// TIA Portal project "1200S7PLC_RS485ModBus_OPCUA" (V19)

(* hardware
DEVICE "S7-1200 station_1"  S7-1200 Station
   slot 0: "Rack_0"  S7-1200 Rack  Rack  V1.0
   slot 1: "PLC_1"  CPU 1212C DC/DC/Rly  6ES7 212-1HE40-0XB0  V4.6
   slot 3: "CB 1241 (RS485)"  CB 1241 (RS485)  6ES7 241-1CH30-1XB0  V1.0
*)

// ===== PLC "PLC_1"  CPU 1212C DC/DC/Rly =====

VAR_GLOBAL   // PLC tag table "Default tag table"
   "System_Byte" AT %MB500 : Byte;
   "FirstScan" AT %M500.0 : Bool;
   "DiagStatusUpdate" AT %M500.1 : Bool;
   "AlwaysTRUE" AT %M500.2 : Bool;
   "AlwaysFALSE" AT %M500.3 : Bool;
   "Clock_Byte" AT %MB501 : Byte;
   "Clock_10Hz" AT %M501.0 : Bool;
   "Clock_5Hz" AT %M501.1 : Bool;
   "Clock_2.5Hz" AT %M501.2 : Bool;
   "Clock_2Hz" AT %M501.3 : Bool;
   "Clock_1.25Hz" AT %M501.4 : Bool;
   "Clock_1Hz" AT %M501.5 : Bool;
   "Clock_0.625Hz" AT %M501.6 : Bool;
   "Clock_0.5Hz" AT %M501.7 : Bool;
   "COMM_LOAD_DONE" AT %M2.0 : Bool;
   "COMM_LOAD_ERROR" AT %M2.1 : Bool;
   "COMM_LOAD_STATUS" AT %MW4 : Word;
   "MASTER_DONE" AT %M2.2 : Bool;
   "MASTER_BUSY" AT %M2.3 : Bool;
   "MASTER_ERROR" AT %M2.4 : Bool;
   "MASTER_STATUS" AT %MW6 : Word;
   "HumidityRaw" AT %MD8 : Real;
   "HumidityReal" AT %MD12 : Real;
   "TemperatureRaw" AT %MD16 : Real;
   "TemperatureReal" AT %MD20 : Real;
END_VAR

DATA_BLOCK "ModbusReadData"   // DB3
{ S7_Optimized_Access := 'FALSE' }
VERSION : 0.1
   VAR
      ModbusSensorData : Array[0..1] of Int;
   END_VAR
BEGIN
END_DATA_BLOCK

FUNCTION "Conversion" : Void   // FC1, LAD
{ S7_Optimized_Access := 'TRUE' }
VERSION : 0.1
BEGIN

REGION Network 1
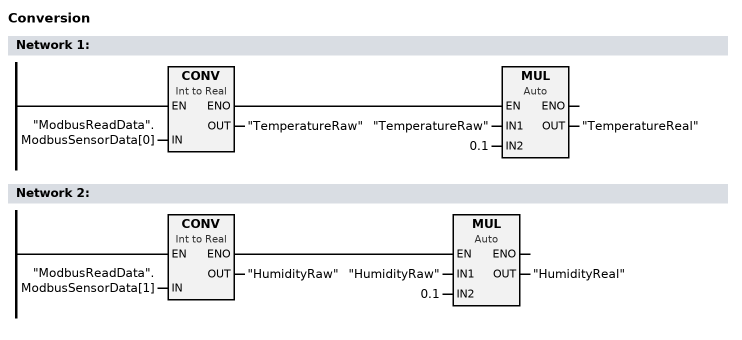
   RUNG wire#powerrail
      { S7_Templates := "[SrcType := Int, DestType := Real]" } Convert(in := "ModbusReadData".ModbusSensorData[0], out => "TemperatureRaw")
      Mul(in1 := "TemperatureRaw", in2 := 0.1, out => "TemperatureReal")
   END_RUNG
   // the same network as SCL:
   "TemperatureRaw" := INT_TO_REAL("ModbusReadData".ModbusSensorData[0]);
   "TemperatureReal" := "TemperatureRaw" * 0.1;
END_REGION

REGION Network 2
   RUNG wire#powerrail
      { S7_Templates := "[SrcType := Int, DestType := Real]" } Convert(in := "ModbusReadData".ModbusSensorData[1], out => "HumidityRaw")
      Mul(in1 := "HumidityRaw", in2 := 0.1, out => "HumidityReal")
   END_RUNG
   // the same network as SCL:
   "HumidityRaw" := INT_TO_REAL("ModbusReadData".ModbusSensorData[1]);
   "HumidityReal" := "HumidityRaw" * 0.1;
END_REGION
END_FUNCTION

ORGANIZATION_BLOCK "Main"   // OB1, LAD, ProgramCycle
TITLE = "Main Program Sweep (Cycle)"
{ S7_Optimized_Access := 'TRUE' }
VERSION : 0.1
   VAR_INPUT
      Initial_Call : Bool;   // Initial call of this OB
      Remanence : Bool;   // =True, if remanent data are available
   END_VAR
BEGIN

REGION Network 1
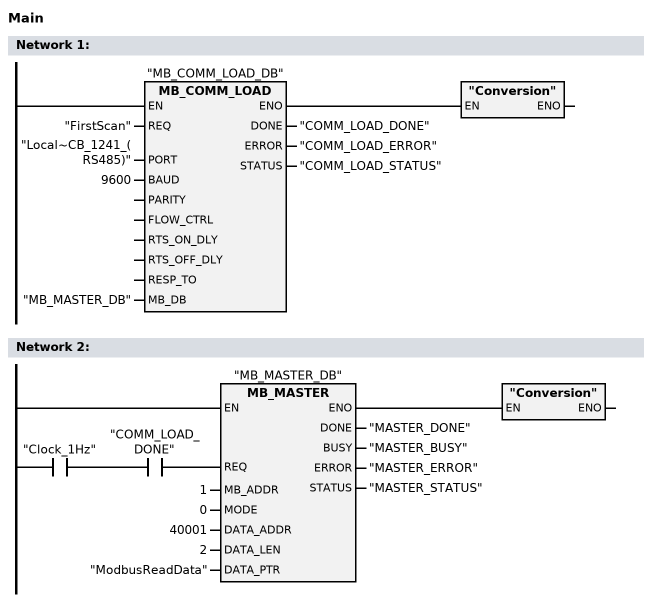
   // ENO of a box is taken as its EN; it also drops when the box reports an error
   "MB_COMM_LOAD_DB"(REQ := "FirstScan",   // MB_COMM_LOAD
                     PORT := "Local~CB_1241_(RS485)",
                     BAUD := 9600,
                     MB_DB := "MB_MASTER_DB",
                     DONE => "COMM_LOAD_DONE",
                     ERROR => "COMM_LOAD_ERROR",
                     STATUS => "COMM_LOAD_STATUS");
   "Conversion"();
END_REGION

REGION Network 2
   // ENO of a box is taken as its EN; it also drops when the box reports an error
   "MB_MASTER_DB"(REQ := "Clock_1Hz" AND "COMM_LOAD_DONE",   // MB_MASTER
                  MB_ADDR := 1,
                  MODE := 0,
                  DATA_ADDR := 40001,
                  DATA_LEN := 2,
                  DATA_PTR := "ModbusReadData",
                  DONE => "MASTER_DONE",
                  BUSY => "MASTER_BUSY",
                  ERROR => "MASTER_ERROR",
                  STATUS => "MASTER_STATUS");
   "Conversion"();
END_REGION
END_ORGANIZATION_BLOCK